FUNCTION_BLOCK HRL_RGB_InitalStateDrive
VAR_INPUT
END_VAR
VAR_OUTPUT
END_VAR
VAR
	HRL_RGB_SRM_InitDrive: AxisControl_MultipleInputSensors;
END_VAR

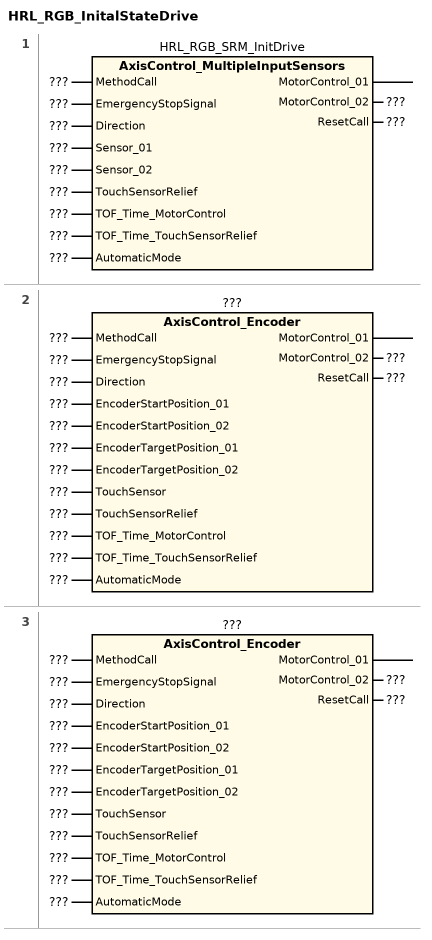
// NETWORK 1
HRL_RGB_SRM_InitDrive(); // AxisControl_MultipleInputSensors

// NETWORK 2
???(); // AxisControl_Encoder

// NETWORK 3
???(); // AxisControl_Encoder

END_FUNCTION_BLOCK

(* stored: Version 1.1.0.1, ProductVersion 3.1.4024.15
   POU HRL_RGB_InitalStateDrive: Id {bd1ed315-dc47-4ef4-bc11-af5370c5e1d4}, SpecialFunc None *)
